// TIA Portal V16 export
// export: Created 2022-04-09T12:19:34.5808705Z, ExportSetting WithDefaults, DisplayName Totally Integrated Automation Portal, DisplayVersion V16 Update 3, DisplayName TIA Portal Version Control Interface, DisplayVersion V16 Update 2, DisplayName TIA Portal Openness, DisplayVersion V16 Update 3, DisplayName STEP 7 Professional, DisplayVersion V16 Update 3, DisplayName STEP 7 Safety, DisplayVersion V16, DisplayName WinCC Professional, DisplayVersion V16 Update 3
DATA_BLOCK "DB39512_Dy_DebugInst2Order"   // DB39512
TITLE = Dynamic DB [DEBUG] — Second Order Response Simulation
{ S7_Optimized_Access := 'TRUE' }
AUTHOR : M_Gledhill
FAMILY : Debug
NAME : Dy_DebugInst2Order
VERSION : 1.1
// PRACTICAL SERIES AUTOMATION LIBRARY (PAL)   —   COPYRIGHT 2020 – M. GLEDHILL (MIT LICENCE)
//                   ———— ◆ ————
// FULL ONLINE DOCUMENTATION IS AVAILABLE AT: https://practicalseries.com/2001-pal/index.html
// stored: AutoNumber false, DBAccessibleFromOPCUA true, IsOnlyStoredInLoadMemory false, IsRetainMemResEnabled false, IsWriteProtectedInAS false, MemoryReserve 100
   VAR
      _DB_Header { ExternalAccessible := 'False'; ExternalVisible := 'False'; ExternalWritable := 'False'} : Array[0..79] of Bool;   // Dynamic DB [DEBUG] — Second Order Response Simulation
      __________0000_0 { ExternalAccessible := 'False'; ExternalVisible := 'False'; ExternalWritable := 'False'} : Bool := false;
      __________0000_1 { ExternalAccessible := 'False'; ExternalVisible := 'False'; ExternalWritable := 'False'} : Bool := false;   // ▀▀▀▀ DB CURRENT REVISION
      revInfo { ExternalWritable := 'False'; S7_SetPoint := 'True'} : "UT01000_St_SysRevision";   // Revision information
      __________0010_0 { ExternalAccessible := 'False'; ExternalVisible := 'False'; ExternalWritable := 'False'} : Bool := false;
      __________0010_1 { ExternalAccessible := 'False'; ExternalVisible := 'False'; ExternalWritable := 'False'} : Bool := false;   // ▀▀▀▀ 2ND ORDER SIMULATION
      SIM001 { ExternalWritable := 'False'} : "UT39512_Dy_DebugInst2Order";   // Simulation 001
   END_VAR
BEGIN
   // _DB_Header[0] : ▄▄▄▄▄▄▄▄▄▄▄▄▄▄▄▄▄▄▄▄▄▄▄▄▄▄▄▄▄▄▄▄▄ ＳＴＡＮＤＡＲＤ ▄▄
   // _DB_Header[2] : TITLE: DEBUG — SECOND ORDER RESPONSE SIMULATION
   // _DB_Header[4] : ▀▀▀▀▀▀▀▀▀▀▀▀▀▀▀▀▀▀▀▀▀▀▀▀▀▀▀▀▀▀▀▀▀▀▀▀▀▀▀▀▀▀▀▀
   // _DB_Header[5] : TYPE: DYNAMIC
   // _DB_Header[6] : ▄▄▄▄▄▄▄▄▄▄▄▄▄▄▄▄▄▄▄▄▄▄▄▄▄▄▄▄▄▄▄▄▄▄▄▄▄▄▄▄▄▄▄▄
   // _DB_Header[8] : This is the dynamic data block associated with the standard DEBUG
   // _DB_Header[9] : Second Order Response Simulation function block:
   // _DB_Header[10] : FC19512_StdDebugInst2Order
   // _DB_Header[12] : The dynamic data holds live data such as calculation variables, simulation elapsed time,
   // _DB_Header[13] : oscillation frequency, status signals and any other information required by the module
   // _DB_Header[15] : Each simulation is given the user data type:
   // _DB_Header[16] : UT39512_Dy_DebugInst2Order
   // _DB_Header[17] : This holds the full set of dynamic data for the simulation
   // _DB_Header[19] : ━━━ ⬙⬙⬙⬙⬙⬙ ━━━
   // _DB_Header[21] : ▄▄▄▄▄▄▄▄▄▄▄▄▄▄▄▄▄▄▄▄▄▄▄▄▄▄▄▄▄▄▄▄▄▄▄▄▄▄▄▄▄▄▄▄
   // _DB_Header[22] : MODIFICATION HISTORY
   // _DB_Header[24] : This is a summary of the recent software modifications made to this block (most recent at top)
   // _DB_Header[26] : ―――――――――――――――――――――――――――――――――――――――――――
   // _DB_Header[27] : DATE REVISION MASTER BRANCH DEV
   // _DB_Header[28] : (nnn.amm) COMMIT TAG (Base ---> Merge) BRANCH Author
   // _DB_Header[29] : ———————————————————————————————————————————
   // _DB_Header[30] : 2022.04.06 001.101 D0010A-000.104 D0010 N/A D010A M. Gledhill
   // _DB_Header[31] : Comments updated and standardised
   // _DB_Header[33] : 2022.03.04 001.000 D0010 D0009 D0010 None M. Gledhill
   // _DB_Header[34] : FC19512 — RELEASED FOR USE
   // _DB_Header[35] : Merge back to master branch
   // _DB_Header[37] : 2022.02.18 000.801 D0009A-000.801 D0009 N/A D0009A M. Gledhill
   // _DB_Header[38] : FC19512 Released for test
   // _DB_Header[40] : 2022.02.18 000.103 D0009A-000.103 D0009 N/A D0009A M. Gledhill
   // _DB_Header[41] : FC19512 Incremental build
   // _DB_Header[43] : 2022.02.02 000.102 D0009A-000.101 D0009 N/A D0009A M. Gledhill
   // _DB_Header[44] : FC19512 Incremental build
   // _DB_Header[45] : ———————————————————————————————————————————
   // _DB_Header[46] : Where: nnn = Major revision
   // _DB_Header[47] : a = Type (1-7 Development, 8 Proving, 9 Qualification, 0 Release)
   // _DB_Header[48] : mm = Minor revision (must be 00 if a = 0)
   // _DB_Header[49] : Block properties version number should be set to nn.a (only one decimal place)
   // _DB_Header[51] : ██████████████ █ █ █ █ END █ █ █ █ ██████████████
   revInfo.REV_BLOCK := 'DB39512';
   revInfo.REV_NUMBER := '001.101';
   revInfo.REV_DATE := '2022-04-06';
   revInfo.REV_AUTHOR := 'M. Gledhill';
END_DATA_BLOCK
